ABB RobotStudio station: 9-Code.rsstnx

Station 9-Code (saved by RobotStudio 25.2.11220.0)
Layout (positions relative to the parent item):
